(*

## Short summary

This class provides assert statements for signed/unsigned integers from 8~64 bit length.
For signed integers use `IntegerAssertions.signed`
For unsigned integers use `IntegerAssertions.unsigned`

.. <legal notes>

legal notes
=================
| SPDX-FileCopyrightText: © 2022 ekvip automation GmbH <info@ekvip.de>
| SPDX-License-Identifier: Apache-2.0
| For details check: Apache-2.0_

.. _Apache-2.0: https://www.apache.org/licenses/LICENSE-2.0

.. </legal notes>

methods aand properties
========================

*)

{attribute 'reflection'}
FUNCTION_BLOCK INTERNAL IntegerAssertions EXTENDS CNM_AbstractObject.Object IMPLEMENTS IIntegerAssertions, IAssertCallBacksetter
VAR
	(* class to handle assert statements for signed integers *)
	signedIntegerAssertions		:SignedIntegerAssertions();
	(* class to handle assert statements for unsigned integers *)
	unsignedIntegerAssertions	:UnsignedIntegerAssertions();
END_VAR

(*

## Short summary
This abstract property returns the class name of the concrete object, 
It's for debugging purpose

.. <legal notes>

legal notes
=================
| SPDX-FileCopyrightText: © 2022 ekvip automation GmbH <info@ekvip.de>
| SPDX-License-Identifier: Apache-2.0
| For details check: Apache-2.0_

.. _Apache-2.0: https://www.apache.org/licenses/LICENSE-2.0

.. </legal notes>

*)

PROPERTY className :CNM_AbstractObject.ClassName
GET
className := 'CNM_AssertionInterfaceLib.IntegerAssertions';
END_GET
END_PROPERTY

(*

## Short summary
This methods is the setter for the callback class if an assertion was false

.. <legal notes>

legal notes
=================
| SPDX-FileCopyrightText: © 2022 ekvip automation GmbH <info@ekvip.de>
| SPDX-License-Identifier: Apache-2.0
| For details check: Apache-2.0_

.. _Apache-2.0: https://www.apache.org/licenses/LICENSE-2.0

.. </legal notes>



*)

METHOD setCallBack
VAR_INPUT
	(* the class that must be informed if an assertion is false *)
	callBack	:IAssertCallBack;  
END_VAR
THIS^.signedIntegerAssertions.setCallBack(callBack);
THIS^.unsignedIntegerAssertions.setCallBack(callBack);
END_METHOD

(*

## Short summary
Returns the interface `ISignedIntegerAssertions` with assert statements for signed integers from 8~64 bit length 

.. <legal notes>

legal notes
=================
| SPDX-FileCopyrightText: © 2022 ekvip automation GmbH <info@ekvip.de>
| SPDX-License-Identifier: Apache-2.0
| For details check: Apache-2.0_

.. _Apache-2.0: https://www.apache.org/licenses/LICENSE-2.0

.. </legal notes>

*)

PROPERTY signed :ISignedIntegerAssertions
GET
signed := THIS^.signedIntegerAssertions;
END_GET
END_PROPERTY

(*

## Short summary
Returns the interface `IUnsignedIntegerAssertions` with assert statements for unsigned integers from 8~64 bit length 

.. <legal notes>

legal notes
=================
| SPDX-FileCopyrightText: © 2022 ekvip automation GmbH <info@ekvip.de>
| SPDX-License-Identifier: Apache-2.0
| For details check: Apache-2.0_

.. _Apache-2.0: https://www.apache.org/licenses/LICENSE-2.0

.. </legal notes>

*)

PROPERTY unsigned :IUnsignedIntegerAssertions
GET
unsigned := THIS^.unsignedIntegerAssertions;
END_GET
END_PROPERTY

END_FUNCTION_BLOCK

(* stored: Version 1.1.0.1, ProductVersion 3.1.4026.12
   POU IntegerAssertions: Id {47fa951a-e2ba-45bf-8ed7-ac4f5e0b6344}, SpecialFunc None
   Property className: Id {ea418b79-6fc3-4065-bdce-46a5da0509af}
   Get Get: Id {bbb004cd-0fe5-48d4-94f8-60777e4a5f29}
   Method setCallBack: Id {6d8c9851-18cf-4094-9661-bd46de76a360}
   Property signed: Id {3b6adec8-1d6a-4a06-b529-89779fee8602}
   Get Get: Id {ee9201e6-5ed3-4340-b7b3-2589e775dccf}
   Property unsigned: Id {684eabc0-bf68-422f-913c-25d616e281b8}
   Get Get: Id {c9df154d-e898-4fe6-a6b8-c070a47ba18f} *)
